// TIA Portal V17 export
// export: Created 2023-12-05T13:40:21.6645103Z, ExportSetting WithDefaults, DisplayName Totally Integrated Automation Portal, DisplayVersion V17, DisplayName TIA Portal Openness, DisplayVersion V17, DisplayName TIA Portal Version Control Interface, DisplayVersion V17, DisplayName SINAMICS Startdrive Advanced, DisplayVersion V17, DisplayName SINAMICS Startdrive G130, G150, S120, S150, SINAMICS MV, S210, DisplayVersion V17, DisplayName SINAMICS Startdrive G110M, G120, G120C, G120D, G120P, G115D, DisplayVersion V17, DisplayName STEP 7 Professional, DisplayVersion V17, DisplayName STEP 7 Safety, DisplayVersion V17, DisplayName WinCC Professional, DisplayVersion V17
FUNCTION "FC514 Move Alarm & IC" : Void   // FC514, LAD
{ S7_Optimized_Access := 'TRUE' }
VERSION : 0.1
// LM Created 2023_06_28
// Movement alarm & Intervention request check
// stored: AutoNumber false, IsIECCheckEnabled false, SetENOAutomatically false, UDAEnableTagReadback false
   VAR_INPUT
      "to WP" : Bool;   // Output Working Position
      "to PP" : Bool;   // Output Parking Position
      "at WP" : Bool;   // Working Position Sensor
      "at PP" : Bool;   // Parking Position Sensor
      "Time for alarm (s)" : USInt;   // Set Time for Alarm
      "to WP/PP manu" : "cylinder";   // Working/Parking Position in Manual
   END_VAR
   VAR_IN_OUT
      "Wp Def" : Bool;   // Working Position Default
      "PP Def" : Bool;   // Parking Position Default
      "Parity Def" : Bool;   // Parity Default
      GeneralStruct : "MoveAlarmGeneral";
      SingleStruct : "MoveAlarmSingle";
   END_VAR
   VAR_TEMP   // added for the SCL form of the ladder/FBD networks
      _w1 : Bool;
      _w2 : Bool;
      _w3 : Bool;
   END_VAR
BEGIN

REGION Network 2: Reset Alarms
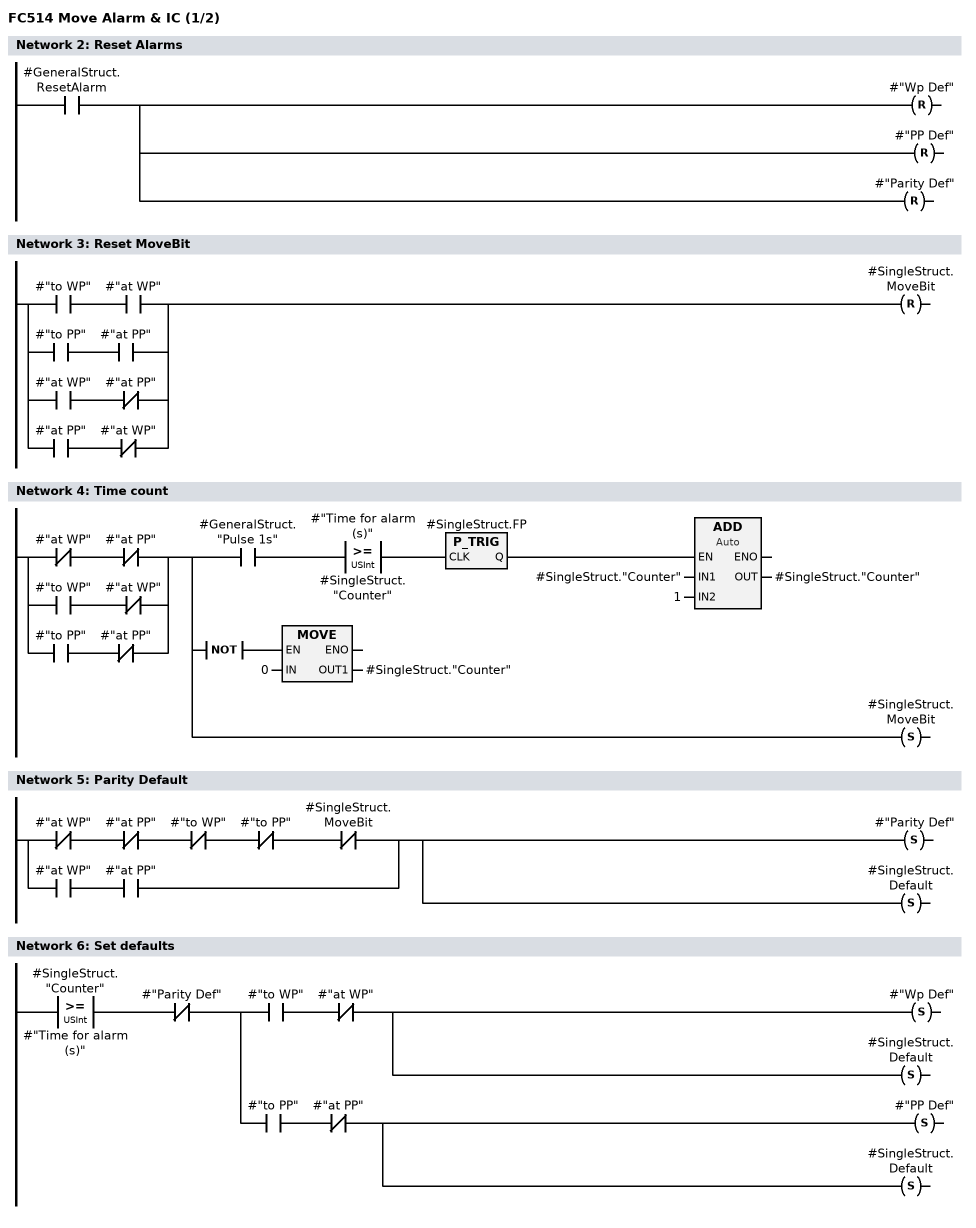
   RUNG wire#powerrail
      Contact( #GeneralStruct.ResetAlarm )
      wire#w1
      R_Coil( #"Wp Def" )
   END_RUNG
   RUNG wire#w1
      R_Coil( #"PP Def" )
   END_RUNG
   RUNG wire#w1
      R_Coil( #"Parity Def" )
   END_RUNG
   // the same network as SCL:
   IF #GeneralStruct.ResetAlarm THEN
       #"Wp Def" := FALSE;
       #"PP Def" := FALSE;
       #"Parity Def" := FALSE;
   END_IF;
END_REGION

REGION Network 3: Reset MoveBit
   RUNG wire#powerrail
      Contact( #"to WP" )
      Contact( #"at WP" )
      wire#w1
      R_Coil( #SingleStruct.MoveBit )
   END_RUNG
   RUNG wire#powerrail
      Contact( #"to PP" )
      Contact( #"at PP" )
   END_RUNG wire#w1
   RUNG wire#powerrail
      Contact( #"at WP" )
      I_Contact( #"at PP" )
   END_RUNG wire#w1
   RUNG wire#powerrail
      Contact( #"at PP" )
      I_Contact( #"at WP" )
   END_RUNG wire#w1
   // the same network as SCL:
   IF (#"to WP" AND #"at WP") OR (#"to PP" AND #"at PP") OR (#"at WP" AND NOT #"at PP") OR (#"at PP" AND NOT #"at WP") THEN
       #SingleStruct.MoveBit := FALSE;
   END_IF;
END_REGION

REGION Network 4: Time count
   RUNG wire#powerrail
      I_Contact( #"at WP" )
      I_Contact( #"at PP" )
      wire#w1
      Contact( #GeneralStruct."Pulse 1s" )
      { S7_Templates := "SrcType := USInt" } GE_Contact(in1 := #"Time for alarm (s)", in2 := #SingleStruct."Counter")
      P_Trig( #SingleStruct.FP )
      Add(in1 := #SingleStruct."Counter", in2 := 1, out => #SingleStruct."Counter")
   END_RUNG
   RUNG wire#powerrail
      Contact( #"to WP" )
      I_Contact( #"at WP" )
   END_RUNG wire#w1
   RUNG wire#powerrail
      Contact( #"to PP" )
      I_Contact( #"at PP" )
   END_RUNG wire#w1
   RUNG wire#w1
      Not()
      Move(in := 0, out1 => #SingleStruct."Counter")
   END_RUNG
   RUNG wire#w1
      S_Coil( #SingleStruct.MoveBit )
   END_RUNG
   // the same network as SCL:
   #_w1 := (NOT #"at WP" AND NOT #"at PP") OR (#"to WP" AND NOT #"at WP") OR (#"to PP" AND NOT #"at PP");
   #_w2 := #_w1 AND #GeneralStruct."Pulse 1s" AND (#"Time for alarm (s)" >= #SingleStruct."Counter");
   #_w3 := #_w2 AND NOT #SingleStruct.FP;   // rising edge
   #SingleStruct.FP := #_w2;
   IF #_w3 THEN #SingleStruct."Counter" := #SingleStruct."Counter" + 1; END_IF;
   IF NOT #_w1 THEN #SingleStruct."Counter" := 0; END_IF;
   IF #_w1 THEN #SingleStruct.MoveBit := TRUE; END_IF;
END_REGION

REGION Network 5: Parity Default
   RUNG wire#powerrail
      I_Contact( #"at WP" )
      I_Contact( #"at PP" )
      I_Contact( #"to WP" )
      I_Contact( #"to PP" )
      I_Contact( #SingleStruct.MoveBit )
      wire#w1
      S_Coil( #"Parity Def" )
   END_RUNG
   RUNG wire#powerrail
      Contact( #"at WP" )
      Contact( #"at PP" )
   END_RUNG wire#w1
   RUNG wire#w1
      S_Coil( #SingleStruct.Default )
   END_RUNG
   // the same network as SCL:
   IF (NOT #"at WP" AND NOT #"at PP" AND NOT #"to WP" AND NOT #"to PP" AND NOT #SingleStruct.MoveBit) OR (#"at WP" AND #"at PP") THEN
       #"Parity Def" := TRUE;
       #SingleStruct.Default := TRUE;
   END_IF;
END_REGION

REGION Network 6: Set defaults
   RUNG wire#powerrail
      { S7_Templates := "SrcType := USInt" } GE_Contact(in1 := #SingleStruct."Counter", in2 := #"Time for alarm (s)")
      I_Contact( #"Parity Def" )
      wire#w1
      Contact( #"to WP" )
      I_Contact( #"at WP" )
      wire#w2
      S_Coil( #"Wp Def" )
   END_RUNG
   RUNG wire#w2
      S_Coil( #SingleStruct.Default )
   END_RUNG
   RUNG wire#w1
      Contact( #"to PP" )
      I_Contact( #"at PP" )
      wire#w3
      S_Coil( #"PP Def" )
   END_RUNG
   RUNG wire#w3
      S_Coil( #SingleStruct.Default )
   END_RUNG
   // the same network as SCL:
   #_w1 := (#SingleStruct."Counter" >= #"Time for alarm (s)") AND NOT #"Parity Def";
   IF #_w1 AND #"to WP" AND NOT #"at WP" THEN
       #"Wp Def" := TRUE;
       #SingleStruct.Default := TRUE;
   END_IF;
   IF #_w1 AND #"to PP" AND NOT #"at PP" THEN
       #"PP Def" := TRUE;
       #SingleStruct.Default := TRUE;
   END_IF;
END_REGION

REGION Network 7: Movement to working in manual mode
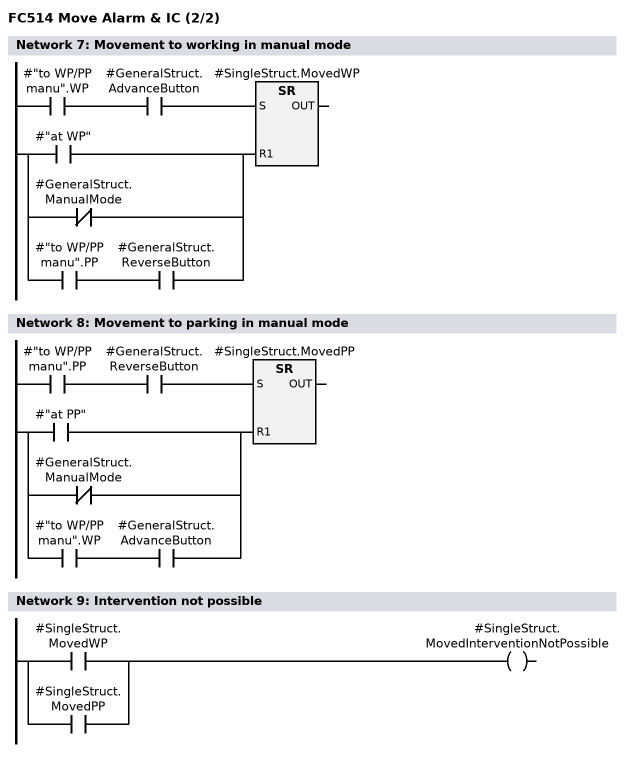
   RUNG wire#powerrail
      Contact( #"to WP/PP manu".WP )
      Contact( #GeneralStruct.AdvanceButton )
      S_SR(operand := #SingleStruct.MovedWP, r1 := wire#w1)
   END_RUNG
   RUNG wire#powerrail
      Contact( #"at WP" )
   END_RUNG wire#w1
   RUNG wire#powerrail
      I_Contact( #GeneralStruct.ManualMode )
   END_RUNG wire#w1
   RUNG wire#powerrail
      Contact( #"to WP/PP manu".PP )
      Contact( #GeneralStruct.ReverseButton )
   END_RUNG wire#w1
   // the same network as SCL:
   IF #"to WP/PP manu".WP AND #GeneralStruct.AdvanceButton THEN
       #SingleStruct.MovedWP := TRUE;   // SR flip-flop
   END_IF;
   IF #"at WP" OR NOT #GeneralStruct.ManualMode OR (#"to WP/PP manu".PP AND #GeneralStruct.ReverseButton) THEN
       #SingleStruct.MovedWP := FALSE;
   END_IF;
END_REGION

REGION Network 8: Movement to parking in manual mode
   RUNG wire#powerrail
      Contact( #"to WP/PP manu".PP )
      Contact( #GeneralStruct.ReverseButton )
      S_SR(operand := #SingleStruct.MovedPP, r1 := wire#w1)
   END_RUNG
   RUNG wire#powerrail
      Contact( #"at PP" )
   END_RUNG wire#w1
   RUNG wire#powerrail
      I_Contact( #GeneralStruct.ManualMode )
   END_RUNG wire#w1
   RUNG wire#powerrail
      Contact( #"to WP/PP manu".WP )
      Contact( #GeneralStruct.AdvanceButton )
   END_RUNG wire#w1
   // the same network as SCL:
   IF #"to WP/PP manu".PP AND #GeneralStruct.ReverseButton THEN
       #SingleStruct.MovedPP := TRUE;   // SR flip-flop
   END_IF;
   IF #"at PP" OR NOT #GeneralStruct.ManualMode OR (#"to WP/PP manu".WP AND #GeneralStruct.AdvanceButton) THEN
       #SingleStruct.MovedPP := FALSE;
   END_IF;
END_REGION

REGION Network 9: Intervention not possible
   RUNG wire#powerrail
      Contact( #SingleStruct.MovedWP )
      wire#w1
      Coil( #SingleStruct.MovedInterventionNotPossible )
   END_RUNG
   RUNG wire#powerrail
      Contact( #SingleStruct.MovedPP )
   END_RUNG wire#w1
   // the same network as SCL:
   #SingleStruct.MovedInterventionNotPossible := #SingleStruct.MovedWP OR #SingleStruct.MovedPP;
END_REGION
END_FUNCTION
